// TIA Portal V20 program export: 2 tag tables, 0 data types, 0 data blocks, 2 code blocks (in call order from the OBs), 0 instance data blocks

VAR_GLOBAL   // PLC tag table "Table de variables standard"
   Clock_Byte AT %MB0 : Byte;
   Clock_10Hz AT %M0.0 : Bool;
   Clock_5Hz AT %M0.1 : Bool;
   "Clock_2.5Hz" AT %M0.2 : Bool;
   Clock_2Hz AT %M0.3 : Bool;
   "Clock_1.25Hz" AT %M0.4 : Bool;
   Clock_1Hz AT %M0.5 : Bool;
   "Clock_0.625Hz" AT %M0.6 : Bool;
   "Clock_0.5Hz" AT %M0.7 : Bool;
   System_Byte AT %MB1 : Byte;
   FirstScan AT %M1.0 : Bool;
   DiagStatusUpdate AT %M1.1 : Bool;
   AlwaysTRUE AT %M1.2 : Bool;
   AlwaysFALSE AT %M1.3 : Bool;
   Tag_1 AT %Q0.0 : Bool;
END_VAR

VAR_GLOBAL   // PLC tag table "Table de variables_1"
   "E0.0" AT %I0.0 : Bool;
   "E0.1" AT %I0.1 : Bool;
   "E0.2" AT %I0.2 : Bool;
   "E0.3" AT %I0.3 : Bool;
   "M2.0" AT %I0.4 : Bool;
   "M2.1" AT %I0.5 : Bool;
END_VAR

ORGANIZATION_BLOCK "Main"   // OB1, LAD, ProgramCycle
TITLE = "Main Program Sweep (Cycle)"
{ S7_Optimized_Access := 'TRUE' }
// stored: SetENOAutomatically false
   VAR_INPUT
      Initial_Call : Bool;
      Remanence : Bool;
   END_VAR
   VAR_TEMP
      temp : Real;
      Position : LReal;
      "Busy_MC-MOVEJOG" : Bool;
      MC_MOVEABSOLUTE : Bool;
   END_VAR
BEGIN

REGION Network 1
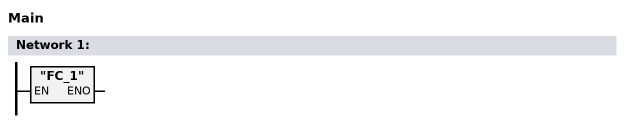
   RUNG wire#powerrail
      "FC_1"()
   END_RUNG
   // the same network as SCL:
   "FC_1"();
END_REGION
END_ORGANIZATION_BLOCK

FUNCTION "FC_1" : Void   // FC1, LAD
{ S7_Optimized_Access := 'TRUE' }
// stored: SetENOAutomatically false
BEGIN

REGION Network 1
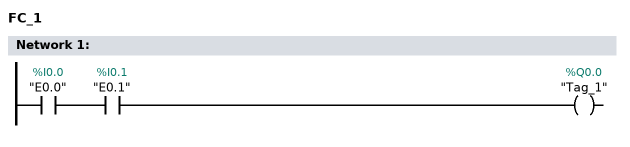
   RUNG wire#powerrail
      Contact( "E0.0" )
      Contact( "E0.1" )
      Coil( "Tag_1" )
   END_RUNG
   // the same network as SCL:
   "Tag_1" := "E0.0" AND "E0.1";
END_REGION
END_FUNCTION
